INTERFACE ITF_Group2_HMI_Connector_Command EXTENDS ITF_BaseGroupElement_HMI_Connector_Command

END_INTERFACE

(* stored: Version 1.1.0.1
   Itf ITF_Group2_HMI_Connector_Command: Id {651cd822-8552-068b-2e41-554f9f9b22d6} *)
